FUNCTION_BLOCK LIMIT_INT (* See LIMIT_ANY *)
  (* Standard: 61131-3 *)
  (* Version 0.0, 2004-12-15, JHC, Rockwell Automation, Converted from SRC format. *)
  (* Compiler header: package fb.rt.plc.select; *)
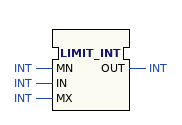
  VAR_INPUT
    MN : INT;
    IN : INT;
    MX : INT;
  END_VAR
  VAR_OUTPUT
    OUT : INT;
  END_VAR
END_FUNCTION_BLOCK
